// TIA Portal V18 export
DATA_BLOCK "FB3-Ratiocheck_DB"   // DB60
VERSION : 0.1
// stored: AutoNumber true, DBAccessibleFromOPCUA true, InstanceOfName FB3-Ratiocheck, InstanceOfType FB
"FB3-Ratiocheck"
   // VAR_INPUT
   //    Dispensing_time : DInt;
   //    "Set Qty in ml" : Real;
   //    "VC1 Pulses" : DInt;
   //    "VC2 Pulses" : DInt;
   //    VC1_impulse : Real;
   //    VC2_impulse : Real;
   //    "Outlet Open  to Pump ON A delay" : DInt;
   //    "Outlet Open  to Pump ON B delay" : DInt;
   //    "Pump Off  to Outlet Close" : DInt;
   //    "Pump Off  to Inlet A Close" : DInt;
   //    "Pump Off  to Inlet B Close" : DInt;
   // END_VAR
   // VAR_OUTPUT
   //    "Volume dispensed" : Real;
   //    "Run time" : Int;
   // END_VAR
   // VAR_IN_OUT
   //    ON_inlet_A : Bool;
   //    ON_inlet_B : Bool;
   //    ON_Pump_A : Bool;
   //    ON_pump_B : Bool;
   //    ON_valve_A : Bool;
   //    ON_valve_B : Bool;
   //    "Start Metering" : Bool;
   //    "Stop metering" : Bool;
   //    "Process running" : Bool;
   //    "process completed" : Bool;
   // END_VAR
   // VAR
   //    "pump A to valveA delay" : Bool;
   //    "Pump B to valve B delay" : Bool;
   //    "Pump Off to mixer off delay_1" : Bool;
   //    "VC1 pulses prev" : DInt;
   //    "VC2 pulses prev" : DInt;
   //    "VC1 pulse generted" : DInt;
   //    "VC2 pulse generated" : DInt;
   //    "Pump A Voulme dispensed" : Real;
   //    "Pump B volume dispensed" : Real;
   //    "Total Volume dispensed" : Real;
   //    "metering started" : Bool;
   //    "metering time in msec" : DInt;
   //    "dispense time elapsed" : Bool;
   // END_VAR
BEGIN
END_DATA_BLOCK
